Staubli VAL3: SplitMoveL.pgx

public program SplitMoveL(string x_sSLine, trsf& x_tr1, trsf& x_trP, bool x_bCut, bool& x_bRes)
  local string l_sChar[2]
  local num l_nData[25]
begin
  x_bRes=false

  if x_sSLine==""
    return
  endIf

  x_sSLine=right(x_sSLine,len(x_sSLine)-len("MOVEL="))

  //解析每一行
  l_sChar[0]=","
  l_sChar[1]="/"

  call SplitNumS(x_sSLine,l_nData,l_sChar,x_bRes)

  if !x_bRes
    return
  endIf

  x_tr1.x=l_nData[0]
  x_tr1.y=l_nData[1]
  x_tr1.z=l_nData[2]
  x_tr1.rx=l_nData[3]
  x_tr1.ry=l_nData[4]
  x_tr1.rz=l_nData[5]



  if !x_bCut

    x_trP.z=l_nData[6]
    x_trP.rx=l_nData[7]
  else
    x_trP.x=l_nData[6]
    x_trP.y=l_nData[7]
    x_trP.z=l_nData[8]
    x_trP.rx=l_nData[9]
    x_trP.ry=l_nData[10]
    //x_trP.rz=l_nData[17]

  endIf




end
